SUBAPPLICATION Automatik (* Subapplication Type *)
  (* Standard: 61499-2 *)
  (* Version 1.0, 2023-01-29, Franz *)
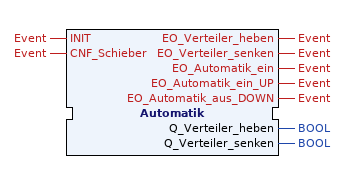
  EVENT_INPUT
    INIT;
    CNF_Schieber;
  END_EVENT
  EVENT_OUTPUT
    EO_Verteiler_heben;
    EO_Verteiler_senken;
    EO_Automatik_ein;
    EO_Automatik_ein_UP;
    EO_Automatik_aus_DOWN;
  END_EVENT
  VAR_OUTPUT
    Q_Verteiler_heben : BOOL;
    Q_Verteiler_senken : BOOL;
  END_VAR
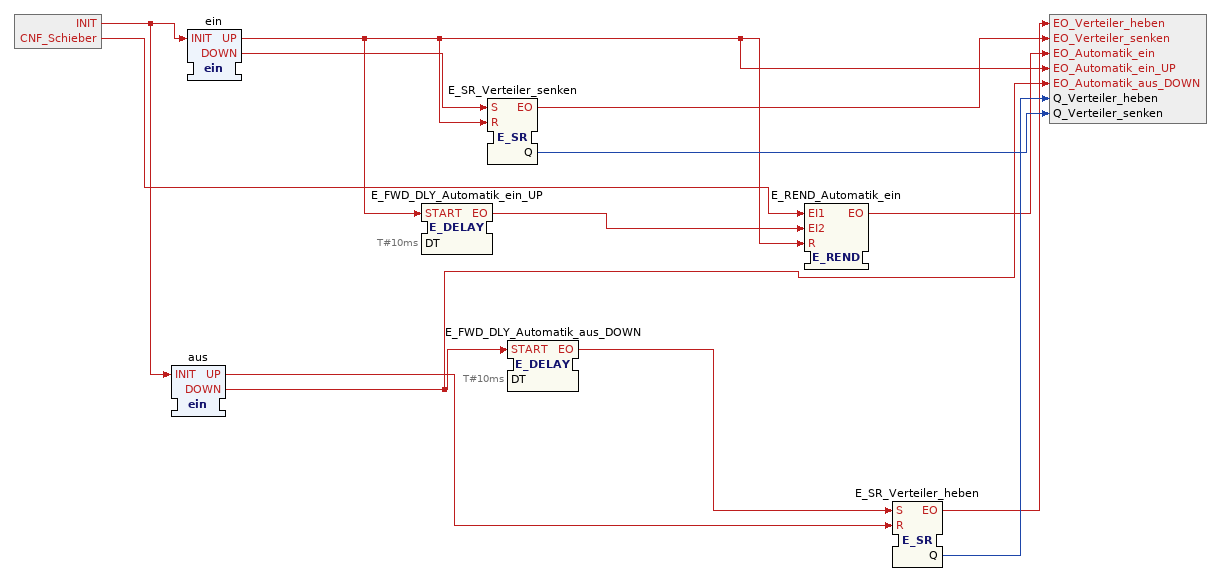
  FBS
    E_SR_Verteiler_heben : E_SR;
    E_SR_Verteiler_senken : E_SR;
    E_REND_Automatik_ein : E_REND;
    E_FWD_DLY_Automatik_ein_UP : E_DELAY(DT := T#10ms);
    E_FWD_DLY_Automatik_aus_DOWN : E_DELAY(DT := T#10ms);
  END_FBS
  SUBAPPS
    ein : ein;
    aus : ein;
  END_SUBAPPS
  EVENT_CONNECTIONS
    E_SR_Verteiler_heben.EO TO EO_Verteiler_heben;
    E_SR_Verteiler_senken.EO TO EO_Verteiler_senken;
    CNF_Schieber TO E_REND_Automatik_ein.EI1;
    E_REND_Automatik_ein.EO TO EO_Automatik_ein;
    E_FWD_DLY_Automatik_ein_UP.EO TO E_REND_Automatik_ein.EI2;
    E_FWD_DLY_Automatik_aus_DOWN.EO TO E_SR_Verteiler_heben.S;
    INIT TO ein.INIT;
    ein.DOWN TO E_SR_Verteiler_senken.S;
    ein.UP TO E_FWD_DLY_Automatik_ein_UP.START;
    ein.UP TO E_SR_Verteiler_senken.R;
    ein.UP TO E_REND_Automatik_ein.R;
    ein.UP TO EO_Automatik_ein_UP;
    INIT TO aus.INIT;
    aus.UP TO E_SR_Verteiler_heben.R;
    aus.DOWN TO E_FWD_DLY_Automatik_aus_DOWN.START;
    aus.DOWN TO EO_Automatik_aus_DOWN;
  END_CONNECTIONS
  DATA_CONNECTIONS
    E_SR_Verteiler_heben.Q TO Q_Verteiler_heben;
    E_SR_Verteiler_senken.Q TO Q_Verteiler_senken;
  END_CONNECTIONS
END_SUBAPPLICATION
